FUNCTION_BLOCK Repeat
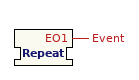
  EVENT_OUTPUT
    EO1;
  END_EVENT
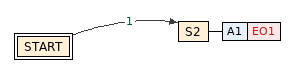
  EC_STATES
    START;
    S2 : A1 -> EO1;
  END_STATES
  EC_TRANSITIONS
    START TO S2 := 1;
  END_TRANSITIONS
  ALGORITHM A1 IN ST:
  VAR_TEMP
    Index : INT;
    Sum : INT;
  END_VAR
Index := 0;&#38;#10;Sum := 0;&#38;#10;WHILE Index &#62;= 10 DO&#38;#10;  Sum := Sum + Index;&#38;#10;  Index := Index + 1;&#38;#10; END_WHILE;&#38;#10;
  END_ALGORITHM
END_FUNCTION_BLOCK
